(* IEC 61131-3 sources: SIGMATEK-Jumag-Utils-Examples/math/Class/comparing, 1 file *)

(* ---- comparing.st ---- *)
(*!
<Class
	Name               = "comparing"
	Revision           = "0.0"
	RealtimeTask       = "false"
	CyclicTask         = "true"
	DefCyclictime      = "100 ms"
	BackgroundTask     = "false"
	Sigmatek           = "false"
	OSInterface        = "false"
	HighPriority       = "false"
	Automatic          = "false"
	UpdateMode         = "Prescan"
	SharedCommandTable = "true"
	Objectsize         = "(284,120)">
	<Channels>
		<Server Name="ClassSvr" Visualized="false" Initialize="false" WriteProtected="true" Retentive="false"/>
	</Channels>
	<Dependencies>
		<Files>
			<File Path=".\Source\math.c"/>
		</Files>
	</Dependencies>
</Class>
*)
comparing : CLASS
  //Servers:
	ClassSvr 	: SvrChCmd_DINT;
  //Clients:
  //Variables:
		isGreaterTest 	: DINT;
		isGreaterEqualTest 	: DINT;
  //Functions:

	FUNCTION VIRTUAL GLOBAL CyWork
		VAR_INPUT
			EAX 	: UDINT;
		END_VAR
		VAR_OUTPUT
			state (EAX) 	: UDINT;
		END_VAR;
  //Tables:
	FUNCTION @STD
		VAR_OUTPUT
			ret_code	: CONFSTATES;
		END_VAR;
	FUNCTION GLOBAL TAB @CT_;
END_CLASS;

Function Global __cdecl isGreater
VAR_INPUT
  CMP1 : REAL;
  CMP2 : REAL;
END_VAR
VAR_OUTPUT
  Q : BOOL;
END_VAR;

Function Global __cdecl isGreaterEqual
VAR_INPUT
  CMP1 : REAL;
  CMP2 : REAL;
END_VAR
VAR_OUTPUT
  Q : BOOL;
END_VAR;

FUNCTION VIRTUAL GLOBAL comparing::CyWork
	VAR_INPUT
		EAX 	: UDINT;
	END_VAR
	VAR_OUTPUT
		state (EAX) 	: UDINT;
	END_VAR

 isGreaterTest := isGreater(CMP1:=10, CMP2:=5);
 isGreaterEqualTest := isGreaterEqual(CMP1:=5, CMP2:=5);

	state := READY;

END_FUNCTION
